(* PLC project mtcs_m1, Institute of Astronomy Onto 0.0.1 *)
(* stored: creationDateTime 2024-10-22T16:57:18.797943, modificationDateTime 2024-10-22T16:57:18.797943 *)

TYPE M1Parts : STRUCT
  inclinometer : M1Inclinometer;  (* Inclinometer *)
  radialSupport : M1RadialSupport;  (* Radial support *)
  axialSupport : M1AxialSupport;  (* Axial support *)
  io : M1M2IO;  (* I/O modules *)
  configManager : ConfigManager;  (* The config manager (to load/save/activate configuration data) *)
END_STRUCT;
END_TYPE

TYPE M1RadialSupportParts : STRUCT
  vacuumRelay : SimpleRelay;  (* Switch Radial vacuum ON to retract the radial pads during mirror manipulations. *)
END_STRUCT;
END_TYPE

TYPE M1M2IOParts : STRUCT
  COU : EtherCatDevice;
  AI1 : EtherCatDevice;
  AI2 : EtherCatDevice;
  AI3 : EtherCatDevice;
  AO1 : EtherCatDevice;
  DO1 : EtherCatDevice;
  RES1 : EtherCatDevice;
  RES2 : EtherCatDevice;
  RES3 : EtherCatDevice;
  PWR1 : EtherCatDevice;
  SSI1 : EtherCatDevice;
  AI4 : EtherCatDevice;
  INC1 : EtherCatDevice;
  P5V1 : EtherCatDevice;
  DO2 : EtherCatDevice;
  DO3 : EtherCatDevice;
  RE1 : EtherCatDevice;
END_STRUCT;
END_TYPE

TYPE M1Processes : STRUCT
  initialize : Process;  (* Start initializing *)
  lock : Process;  (* Lock the system *)
  unlock : Process;  (* Unlock the system *)
  changeOperatingState : ChangeOperatingStateProcess;  (* Change the operating state (e.g. AUTO, MANUAL, ...) *)
END_STRUCT;
END_TYPE

TYPE M1RadialSupportProcesses : STRUCT
  changePressureSetpoint : ChangeSetpointProcess;  (* Change a pressure setpoint, in Bar *)
  changePressureSetpointState : ChangeOperatingStateProcess;  (* Change the operating state of the pressure setpoint only *)
END_STRUCT;
END_TYPE

TYPE M1AxialSupportProcesses : STRUCT
  changePressureSetpoint : ChangeSetpointProcess;  (* Change a pressure setpoint, in Bar *)
  changePressureSetpointState : ChangeOperatingStateProcess;  (* Change the operating state of the pressure setpoint only *)
END_STRUCT;
END_TYPE

TYPE M1Statuses : STRUCT
  initializationStatus : InitializationStatus;
  healthStatus : HealthStatus;
  busyStatus : BusyStatus;
  operatingStatus : OperatingStatus;
END_STRUCT;
END_TYPE

TYPE M1InclinometerStatuses : STRUCT
  healthStatus : HealthStatus;  (* Is the inclinometer elevation trustworthy? *)
END_STRUCT;
END_TYPE

TYPE M1RadialSupportStatuses : STRUCT
  pressureSetpointStatus : OperatingStatus;  (* Operating status of the radial pressure setpoint *)
  healthStatus : HealthStatus;
  busyStatus : BusyStatus;
END_STRUCT;
END_TYPE

TYPE M1AxialSupportStatuses : STRUCT
  pressureSetpointStatus : OperatingStatus;  (* Operating status of the radial pressure setpoint *)
  healthStatus : HealthStatus;
  busyStatus : BusyStatus;
END_STRUCT;
END_TYPE

TYPE M1M2IOStatuses : STRUCT
  healthStatus : HealthStatus;  (* Is the I/O in a healthy state? *)
END_STRUCT;
END_TYPE

TYPE M1Config : STRUCT
  radialSupport : M1RadialSupportConfig;  (* Radial support *)
  axialSupport : M1AxialSupportConfig;  (* Axial support *)
  pneumaticSupplySensorFullScale : LREAL;  (* Sensor full scale range, in Bar *)
  pneumaticSupplyPressure : MeasurementConfig;  (* Pneumatic supply pressure config, in Bar *)
  inclinometerVoltage : MeasurementConfig;  (* Inclinometer voltage measuremennt config, in Volts *)
END_STRUCT;
END_TYPE

TYPE M1RadialSupportConfig : STRUCT
  regulatorPressure : MeasurementConfig;  (* Regulator pressure config, in Bar *)
  mirrorPressure : MeasurementConfig;  (* Regulator pressure config, in Bar *)
  regulatorPressureSensorFullScale : LREAL;  (* Sensor full scale range, in Bar *)
  mirrorPressureSensorFullScale : LREAL;  (* Sensor full scale range, in Bar *)
  correctionCoefficient : LREAL;  (* Correction coefficient for radial pressure *)
  controllerLimitMax : LREAL;  (* Maximum output of the controller, in Bar *)
  controllerLimitMin : LREAL;  (* Minimum output of the controller, in Bar *)
  pressureRegulatorRange : LREAL;  (* Pressure regulator range, in Bar *)
END_STRUCT;
END_TYPE

TYPE M1AxialSupportConfig : STRUCT
  regulatorPressure : MeasurementConfig;  (* Regulator pressure config, in Bar *)
  mirrorPressure : MeasurementConfig;  (* Regulator pressure config, in Bar *)
  mirrorSouthForce : MeasurementConfig;  (* Mirror south force config, in decaNewton *)
  mirrorNorthEastForce : MeasurementConfig;  (* Mirror north east force config, in decaNewton *)
  mirrorNorthWestForce : MeasurementConfig;  (* Mirror north west force config, in decaNewton *)
  mirrorAverageForce : MeasurementConfig;  (* Mirror moving average force config, in decaNewton *)
  regulatorPressureSensorFullScale : LREAL;  (* Sensor full scale range, in Bar *)
  mirrorPressureSensorFullScale : LREAL;  (* Sensor full scale range, in Bar *)
  correctionCoefficient : LREAL;  (* Correction coefficient for axial pressure *)
  controllerKp : LREAL;  (* Proportional factor (gain) of the PI controller *)
  controllerTn : LREAL;  (* Integral time factor of the PI controller. in seconds *)
  controllerLimitMax : LREAL;  (* Maximum output of the controller, in Bar *)
  controllerLimitMin : LREAL;  (* Minimum output of the controller, in Bar *)
  pressureRegulatorRange : LREAL;  (* Pressure regulator range, in Bar *)
END_STRUCT;
END_TYPE

FUNCTION_BLOCK SM_M1
  VAR_INPUT
    {attribute 'OPC.UA.DA' := '1'}
    {attribute 'OPC.UA.DA.Access' := '1'}
    editableConfig : M1Config;  (* Editable configuration of the M1 subsystem *)
  END_VAR
  VAR_OUTPUT
    {attribute 'OPC.UA.DA' := '1'}
    {attribute 'OPC.UA.DA.Access' := '1'}
    actualStatus : STRING;  (* Current status description *)
    previousStatus : STRING;  (* Previous status description *)
    {attribute 'OPC.UA.DA' := '1'}
    {attribute 'OPC.UA.DA.Access' := '1'}
    config : M1Config;  (* Active configuration of the M1 subsystem *)
    {attribute 'OPC.UA.DA' := '1'}
    {attribute 'OPC.UA.DA.Access' := '1'}
    pneumaticSupplyPressure : PressureMeasurement;  (* Pressure measurement of the pneumatic supply *)
    statuses : M1Statuses;  (* Statuses of the state machine *)
    parts : M1Parts;  (* Parts of the state machine *)
    processes : M1Processes;  (* Processes of the state machine *)
  END_VAR
  VAR_IN_OUT
    {attribute 'OPC.UA.DA' := '0'}
    operatorStatus : OperatorStatus;  (* Shared operator status *)
    {attribute 'OPC.UA.DA' := '0'}
    tubeAngleMeasurement : TelemetryAccelerometer;  (* Accelerometer box angle measurement *)
  END_VAR

            pneumaticSupplyPressure(
    config := config.pneumaticSupplyPressure,
    conversionFactor := config.pneumaticSupplySensorFullScale / 32768.0);
parts.inclinometer( config := config.inclinometerVoltage );
parts.radialSupport(
    config := config.radialSupport,
    inclinometer := parts.inclinometer,
    operatorStatus := operatorStatus,
    operatingStatus := statuses.operatingStatus);
parts.axialSupport(
    config := config.axialSupport,
    inclinometer := parts.inclinometer,
    operatorStatus := operatorStatus,
    operatingStatus := statuses.operatingStatus,
    tubeAngle := tubeAngleMeasurement.averageYAngle);
parts.io();
parts.configManager( isEnabled := operatorStatus.tech );
statuses.initializationStatus();
statuses.healthStatus(
    isGood := parts.radialSupport.statuses.healthStatus.isGood AND (parts.axialSupport.statuses.healthStatus.isGood AND (parts.io.statuses.healthStatus.isGood AND parts.configManager.statuses.healthStatus.isGood)),
    hasWarning := parts.radialSupport.statuses.healthStatus.hasWarning OR (parts.axialSupport.statuses.healthStatus.hasWarning OR (parts.io.statuses.healthStatus.hasWarning OR parts.configManager.statuses.healthStatus.hasWarning)));
statuses.busyStatus( isBusy := statuses.initializationStatus.initializing OR (parts.radialSupport.statuses.busyStatus.busy OR (parts.axialSupport.statuses.busyStatus.busy OR parts.configManager.statuses.busyStatus.busy)) );
statuses.operatingStatus( superState := statuses.initializationStatus.initialized );
processes.initialize( isEnabled := statuses.initializationStatus.shutdown OR (statuses.initializationStatus.initializingFailed OR statuses.initializationStatus.initialized) );
processes.lock( isEnabled := operatorStatus.tech AND statuses.initializationStatus.initialized );
processes.unlock( isEnabled := operatorStatus.tech AND statuses.initializationStatus.locked );
processes.changeOperatingState( isEnabled := statuses.busyStatus.idle AND (statuses.initializationStatus.initialized AND operatorStatus.tech) );

          

{attribute 'TcRpcEnable' := '1'}
METHOD initialize : RequestResults
                  initialize := THIS^.processes.initialize.request();

                
END_METHOD

{attribute 'TcRpcEnable' := '1'}
METHOD lock : RequestResults
                  lock := THIS^.processes.lock.request();

                
END_METHOD

{attribute 'TcRpcEnable' := '1'}
METHOD unlock : RequestResults
                  unlock := THIS^.processes.unlock.request();

                
END_METHOD

{attribute 'TcRpcEnable' := '1'}
METHOD changeOperatingState : RequestResults
  VAR_INPUT
    state : OperatingStates;
  END_VAR
                  changeOperatingState := THIS^.processes.changeOperatingState.request( state := state );

                
END_METHOD

{attribute 'TcRpcEnable' := '1'}
METHOD _log : BOOL
  VAR_INPUT
    name : STRING;  (* Name of this function block instance *)
  END_VAR
  VAR_IN_OUT
    buffer : LogBuffer;  (* Buffer to write all logging to *)
  END_VAR
  VAR
    subBuffer : LogBuffer;  (* Temporary buffer to write logging by parts (sub-statemachines) to *)
  END_VAR
                  THIS^.parts.inclinometer._log(
    name := 'inclinometer',
    buffer := subBuffer);
THIS^.parts.radialSupport._log(
    name := 'radialSupport',
    buffer := subBuffer);
THIS^.parts.axialSupport._log(
    name := 'axialSupport',
    buffer := subBuffer);
THIS^.parts.io._log(
    name := 'io',
    buffer := subBuffer);
THIS^.parts.configManager._log(
    name := 'configManager',
    buffer := subBuffer);
THIS^.processes.initialize._log(
    name := 'processes.initialize',
    buffer := subBuffer);
THIS^.processes.lock._log(
    name := 'processes.lock',
    buffer := subBuffer);
THIS^.processes.unlock._log(
    name := 'processes.unlock',
    buffer := subBuffer);
THIS^.processes.changeOperatingState._log(
    name := 'processes.changeOperatingState',
    buffer := subBuffer);
LOGGER(
    name := name,
    actualStatus := THIS^.actualStatus,
    previousStatus := THIS^.previousStatus,
    buffer := buffer,
    subBuffer := subBuffer,
    pHealthStatus := ADR(THIS^.statuses.healthStatus),
    pBusyStatus := ADR(THIS^.statuses.busyStatus));

                
END_METHOD
END_FUNCTION_BLOCK

FUNCTION_BLOCK SM_M1Inclinometer
  VAR_INPUT
    {attribute 'OPC.UA.DA' := '1'}
    {attribute 'OPC.UA.DA.Access' := '1'}
    voltageMeasurement : VoltageMeasurement;  (* Measured voltage *)
  END_VAR
  VAR_OUTPUT
    {attribute 'OPC.UA.DA' := '1'}
    {attribute 'OPC.UA.DA.Access' := '1'}
    actualStatus : STRING;  (* Current status description *)
    previousStatus : STRING;  (* Previous status description *)
    {attribute 'OPC.UA.DA' := '1'}
    {attribute 'OPC.UA.DA.Access' := '1'}
    actualElevation : AngularPosition;  (* Elevation actual value *)
    {attribute 'OPC.UA.DA' := '1'}
    {attribute 'OPC.UA.DA.Access' := '1'}
    averageElevation : AngularPosition;  (* Elevation average value *)
    statuses : M1InclinometerStatuses;  (* Statuses of the state machine *)
  END_VAR
  VAR_IN_OUT
    {attribute 'OPC.UA.DA' := '0'}
    config : MeasurementConfig;  (* Reference to the config *)
  END_VAR

            voltageMeasurement(
    config := config,
    conversionFactor := 10.0 / 32768.0);
statuses.healthStatus(
    isGood := voltageMeasurement.statuses.healthStatus.isGood,
    hasWarning := voltageMeasurement.statuses.healthStatus.hasWarning);

          

{attribute 'TcRpcEnable' := '1'}
METHOD _log : BOOL
  VAR_INPUT
    name : STRING;  (* Name of this function block instance *)
  END_VAR
  VAR_IN_OUT
    buffer : LogBuffer;  (* Buffer to write all logging to *)
  END_VAR
  VAR
    subBuffer : LogBuffer;  (* Temporary buffer to write logging by parts (sub-statemachines) to *)
  END_VAR
                  LOGGER(
    name := name,
    actualStatus := THIS^.actualStatus,
    previousStatus := THIS^.previousStatus,
    buffer := buffer,
    subBuffer := subBuffer,
    pHealthStatus := ADR(THIS^.statuses.healthStatus));

                
END_METHOD
END_FUNCTION_BLOCK

FUNCTION_BLOCK SM_M1RadialSupport
  VAR_INPUT
    {attribute 'OPC.UA.DA' := '0'}
    pressureSetpointOutput AT %Q* : INT;  (* Output value *)
  END_VAR
  VAR_OUTPUT
    {attribute 'OPC.UA.DA' := '1'}
    {attribute 'OPC.UA.DA.Access' := '1'}
    actualStatus : STRING;  (* Current status description *)
    previousStatus : STRING;  (* Previous status description *)
    {attribute 'OPC.UA.DA' := '1'}
    {attribute 'OPC.UA.DA.Access' := '1'}
    regulatorPressure : PressureMeasurement;  (* Pressure measurement at the regulator *)
    {attribute 'OPC.UA.DA' := '1'}
    {attribute 'OPC.UA.DA.Access' := '1'}
    mirrorPressure : PressureMeasurement;  (* Pressure measurement at the mirror *)
    {attribute 'OPC.UA.DA' := '1'}
    {attribute 'OPC.UA.DA.Access' := '1'}
    actualPressureSetpoint : Pressure;  (* Pressure setpoint actually used *)
    {attribute 'OPC.UA.DA' := '1'}
    {attribute 'OPC.UA.DA.Access' := '1'}
    autoPressureSetpoint : Pressure;  (* Pressure setpoint in AUTO mode *)
    {attribute 'OPC.UA.DA' := '1'}
    {attribute 'OPC.UA.DA.Access' := '1'}
    manualPressureSetpoint : Pressure;  (* Pressure setpoint in MANUAL mode *)
    statuses : M1RadialSupportStatuses;  (* Statuses of the state machine *)
    parts : M1RadialSupportParts;  (* Parts of the state machine *)
    processes : M1RadialSupportProcesses;  (* Processes of the state machine *)
  END_VAR
  VAR_IN_OUT
    {attribute 'OPC.UA.DA' := '0'}
    config : M1RadialSupportConfig;
    {attribute 'OPC.UA.DA' := '0'}
    inclinometer : M1Inclinometer;
    {attribute 'OPC.UA.DA' := '0'}
    operatorStatus : OperatorStatus;
    {attribute 'OPC.UA.DA' := '0'}
    operatingStatus : OperatingStatus;
  END_VAR

            regulatorPressure(
    config := config.regulatorPressure,
    conversionFactor := config.regulatorPressureSensorFullScale / 32768.0);
mirrorPressure(
    config := config.mirrorPressure,
    conversionFactor := config.mirrorPressureSensorFullScale / 32768.0);
parts.vacuumRelay( isEnabled := statuses.busyStatus.idle AND (operatingStatus.manual AND operatorStatus.tech) );
statuses.pressureSetpointStatus();
statuses.healthStatus(
    isGood := (processes.changePressureSetpointState.statuses.healthStatus.isGood AND (processes.changePressureSetpoint.statuses.healthStatus.isGood AND regulatorPressure.statuses.healthStatus.isGood)) AND (mirrorPressure.statuses.healthStatus.isGood OR mirrorPressure.statuses.enabledStatus.disabled),
    hasWarning := (processes.changePressureSetpointState.statuses.healthStatus.hasWarning OR (processes.changePressureSetpoint.statuses.healthStatus.hasWarning OR (regulatorPressure.statuses.healthStatus.hasWarning OR mirrorPressure.statuses.healthStatus.hasWarning))) OR parts.vacuumRelay.digitalOutput);
statuses.busyStatus( isBusy := processes.changePressureSetpointState.statuses.busyStatus.busy OR (processes.changePressureSetpoint.statuses.busyStatus.busy OR parts.vacuumRelay.statuses.busyStatus.busy) );
processes.changePressureSetpoint( isEnabled := parts.vacuumRelay.isEnabled );
processes.changePressureSetpointState( isEnabled := parts.vacuumRelay.isEnabled );

          

{attribute 'TcRpcEnable' := '1'}
METHOD changePressureSetpoint : RequestResults
  VAR_INPUT
    setpoint : LREAL;
  END_VAR
                  changePressureSetpoint := THIS^.processes.changePressureSetpoint.request( setpoint := setpoint );

                
END_METHOD

{attribute 'TcRpcEnable' := '1'}
METHOD changePressureSetpointState : RequestResults
  VAR_INPUT
    state : OperatingStates;
  END_VAR
                  changePressureSetpointState := THIS^.processes.changePressureSetpointState.request( state := state );

                
END_METHOD

{attribute 'TcRpcEnable' := '1'}
METHOD _log : BOOL
  VAR_INPUT
    name : STRING;  (* Name of this function block instance *)
  END_VAR
  VAR_IN_OUT
    buffer : LogBuffer;  (* Buffer to write all logging to *)
  END_VAR
  VAR
    subBuffer : LogBuffer;  (* Temporary buffer to write logging by parts (sub-statemachines) to *)
  END_VAR
                  THIS^.parts.vacuumRelay._log(
    name := 'vacuumRelay',
    buffer := subBuffer);
THIS^.processes.changePressureSetpoint._log(
    name := 'processes.changePressureSetpoint',
    buffer := subBuffer);
THIS^.processes.changePressureSetpointState._log(
    name := 'processes.changePressureSetpointState',
    buffer := subBuffer);
LOGGER(
    name := name,
    actualStatus := THIS^.actualStatus,
    previousStatus := THIS^.previousStatus,
    buffer := buffer,
    subBuffer := subBuffer,
    pHealthStatus := ADR(THIS^.statuses.healthStatus),
    pBusyStatus := ADR(THIS^.statuses.busyStatus));

                
END_METHOD
END_FUNCTION_BLOCK

FUNCTION_BLOCK SM_M1AxialSupport
  VAR_INPUT
    {attribute 'OPC.UA.DA' := '0'}
    pressureSetpointOutput AT %Q* : INT;  (* Output value *)
  END_VAR
  VAR_OUTPUT
    {attribute 'OPC.UA.DA' := '1'}
    {attribute 'OPC.UA.DA.Access' := '1'}
    actualStatus : STRING;  (* Current status description *)
    previousStatus : STRING;  (* Previous status description *)
    {attribute 'OPC.UA.DA' := '1'}
    {attribute 'OPC.UA.DA.Access' := '1'}
    regulatorPressure : PressureMeasurement;  (* Pressure measurement at the regulator *)
    {attribute 'OPC.UA.DA' := '1'}
    {attribute 'OPC.UA.DA.Access' := '1'}
    mirrorPressure : PressureMeasurement;  (* Pressure measurement at the mirror *)
    {attribute 'OPC.UA.DA' := '1'}
    {attribute 'OPC.UA.DA.Access' := '1'}
    mirrorSouthForce : ForceMeasurement;  (* Force measurement South (SO) *)
    {attribute 'OPC.UA.DA' := '1'}
    {attribute 'OPC.UA.DA.Access' := '1'}
    mirrorNorthEastForce : ForceMeasurement;  (* Force measurement North East (NE) *)
    {attribute 'OPC.UA.DA' := '1'}
    {attribute 'OPC.UA.DA.Access' := '1'}
    mirrorNorthWestForce : ForceMeasurement;  (* Force measurement North West (NW) *)
    {attribute 'OPC.UA.DA' := '1'}
    {attribute 'OPC.UA.DA.Access' := '1'}
    mirrorAverageForce : ForceMeasurement;  (* Average of SO, NE and NW *)
    {attribute 'OPC.UA.DA' := '1'}
    {attribute 'OPC.UA.DA.Access' := '1'}
    actualPressureSetpoint : Pressure;  (* Pressure setpoint actually used *)
    {attribute 'OPC.UA.DA' := '1'}
    {attribute 'OPC.UA.DA.Access' := '1'}
    autoPressureSetpoint : Pressure;  (* Pressure setpoint in AUTO mode *)
    {attribute 'OPC.UA.DA' := '1'}
    {attribute 'OPC.UA.DA.Access' := '1'}
    manualPressureSetpoint : Pressure;  (* Pressure setpoint in MANUAL mode *)
    {attribute 'OPC.UA.DA' := '1'}
    {attribute 'OPC.UA.DA.Access' := '1'}
    controllerSetpoint : Force;  (* Force setpoint of the controller *)
    statuses : M1AxialSupportStatuses;  (* Statuses of the state machine *)
    processes : M1AxialSupportProcesses;  (* Processes of the state machine *)
  END_VAR
  VAR_IN_OUT
    {attribute 'OPC.UA.DA' := '0'}
    config : M1AxialSupportConfig;
    {attribute 'OPC.UA.DA' := '0'}
    inclinometer : M1Inclinometer;
    {attribute 'OPC.UA.DA' := '0'}
    operatorStatus : OperatorStatus;
    {attribute 'OPC.UA.DA' := '0'}
    operatingStatus : OperatingStatus;
    {attribute 'OPC.UA.DA' := '0'}
    tubeAngle : AngularPosition;
  END_VAR

            regulatorPressure(
    config := config.regulatorPressure,
    conversionFactor := config.regulatorPressureSensorFullScale / 32768.0);
mirrorPressure(
    config := config.mirrorPressure,
    conversionFactor := config.mirrorPressureSensorFullScale / 32768.0);
mirrorSouthForce(
    config := config.mirrorSouthForce,
    conversionFactor := (-200.0 * 20.0) / 2147483648.0);
mirrorNorthEastForce(
    config := config.mirrorNorthEastForce,
    conversionFactor := (-200.0 * 20.0) / 2147483648.0);
mirrorNorthWestForce(
    config := config.mirrorNorthWestForce,
    conversionFactor := (-200.0 * 20.0) / 2147483648.0);
mirrorAverageForce(
    config := config.mirrorAverageForce,
    conversionFactor := (-200.0 * 20.0) / 2147483648.0);
statuses.pressureSetpointStatus();
statuses.healthStatus(
    isGood := (processes.changePressureSetpointState.statuses.healthStatus.isGood AND (processes.changePressureSetpoint.statuses.healthStatus.isGood AND (regulatorPressure.statuses.healthStatus.isGood AND mirrorAverageForce.statuses.healthStatus.isGood))) AND (mirrorPressure.statuses.healthStatus.isGood OR mirrorPressure.statuses.enabledStatus.disabled),
    hasWarning := processes.changePressureSetpointState.statuses.healthStatus.hasWarning OR (processes.changePressureSetpoint.statuses.healthStatus.hasWarning OR (regulatorPressure.statuses.healthStatus.hasWarning OR (mirrorPressure.statuses.healthStatus.hasWarning OR mirrorAverageForce.statuses.healthStatus.hasWarning))));
statuses.busyStatus( isBusy := processes.changePressureSetpointState.statuses.busyStatus.busy OR processes.changePressureSetpoint.statuses.busyStatus.busy );
processes.changePressureSetpoint( isEnabled := statuses.busyStatus.idle AND (operatingStatus.manual AND operatorStatus.tech) );
processes.changePressureSetpointState( isEnabled := statuses.busyStatus.idle AND (operatingStatus.manual AND operatorStatus.tech) );

          

{attribute 'TcRpcEnable' := '1'}
METHOD changePressureSetpoint : RequestResults
  VAR_INPUT
    setpoint : LREAL;
  END_VAR
                  changePressureSetpoint := THIS^.processes.changePressureSetpoint.request( setpoint := setpoint );

                
END_METHOD

{attribute 'TcRpcEnable' := '1'}
METHOD changePressureSetpointState : RequestResults
  VAR_INPUT
    state : OperatingStates;
  END_VAR
                  changePressureSetpointState := THIS^.processes.changePressureSetpointState.request( state := state );

                
END_METHOD

{attribute 'TcRpcEnable' := '1'}
METHOD _log : BOOL
  VAR_INPUT
    name : STRING;  (* Name of this function block instance *)
  END_VAR
  VAR_IN_OUT
    buffer : LogBuffer;  (* Buffer to write all logging to *)
  END_VAR
  VAR
    subBuffer : LogBuffer;  (* Temporary buffer to write logging by parts (sub-statemachines) to *)
  END_VAR
                  THIS^.processes.changePressureSetpoint._log(
    name := 'processes.changePressureSetpoint',
    buffer := subBuffer);
THIS^.processes.changePressureSetpointState._log(
    name := 'processes.changePressureSetpointState',
    buffer := subBuffer);
LOGGER(
    name := name,
    actualStatus := THIS^.actualStatus,
    previousStatus := THIS^.previousStatus,
    buffer := buffer,
    subBuffer := subBuffer,
    pHealthStatus := ADR(THIS^.statuses.healthStatus),
    pBusyStatus := ADR(THIS^.statuses.busyStatus));

                
END_METHOD
END_FUNCTION_BLOCK

FUNCTION_BLOCK SM_M1M2IO
  VAR_OUTPUT
    {attribute 'OPC.UA.DA' := '1'}
    {attribute 'OPC.UA.DA.Access' := '1'}
    actualStatus : STRING;  (* Current status description *)
    previousStatus : STRING;  (* Previous status description *)
    statuses : M1M2IOStatuses;  (* Statuses of the state machine *)
    parts : M1M2IOParts;  (* Parts of the state machine *)
  END_VAR

            parts.COU(
    id := 'M1M2:COU',
    typeId := 'EK1101');
parts.AI1(
    id := 'M1M2:AI1',
    typeId := 'EL3102');
parts.AI2(
    id := 'M1M2:AI2',
    typeId := 'EL3204');
parts.AI3(
    id := 'M1M2:AI3',
    typeId := 'EL3204');
parts.AO1(
    id := 'M1M2:AO1',
    typeId := 'EL4022');
parts.DO1(
    id := 'M1M2:DO1',
    typeId := 'EL2024');
parts.RES1(
    id := 'M1M2:RES1',
    typeId := 'EL3351');
parts.RES2(
    id := 'M1M2:RES2',
    typeId := 'EL3351');
parts.RES3(
    id := 'M1M2:RES3',
    typeId := 'EL3351');
parts.PWR1(
    id := 'M1M2:PWR1',
    typeId := 'EL9410');
parts.SSI1(
    id := 'M1M2:SSI1',
    typeId := 'EL5001');
parts.AI4(
    id := 'M1M2:AI4',
    typeId := 'EL3164');
parts.INC1(
    id := 'M1M2:INC1',
    typeId := 'ES5101');
parts.P5V1(
    id := 'M1M2:P5V1',
    typeId := 'EL9505');
parts.DO2(
    id := 'M1M2:DO2',
    typeId := 'EL2124');
parts.DO3(
    id := 'M1M2:DO3',
    typeId := 'EL2124');
parts.RE1(
    id := 'M1M2:RE1',
    typeId := 'EL2622');
statuses.healthStatus( isGood := parts.COU.statuses.healthStatus.isGood AND (parts.AI1.statuses.healthStatus.isGood AND (parts.AI2.statuses.healthStatus.isGood AND (parts.AI3.statuses.healthStatus.isGood AND (parts.AO1.statuses.healthStatus.isGood AND (parts.DO1.statuses.healthStatus.isGood AND (parts.RES1.statuses.healthStatus.isGood AND (parts.RES2.statuses.healthStatus.isGood AND (parts.RES3.statuses.healthStatus.isGood AND (parts.PWR1.statuses.healthStatus.isGood AND (parts.SSI1.statuses.healthStatus.isGood AND (parts.AI4.statuses.healthStatus.isGood AND (parts.INC1.statuses.healthStatus.isGood AND (parts.P5V1.statuses.healthStatus.isGood AND (parts.DO2.statuses.healthStatus.isGood AND (parts.DO3.statuses.healthStatus.isGood AND parts.RE1.statuses.healthStatus.isGood))))))))))))))) );

          

{attribute 'TcRpcEnable' := '1'}
METHOD _log : BOOL
  VAR_INPUT
    name : STRING;  (* Name of this function block instance *)
  END_VAR
  VAR_IN_OUT
    buffer : LogBuffer;  (* Buffer to write all logging to *)
  END_VAR
  VAR
    subBuffer : LogBuffer;  (* Temporary buffer to write logging by parts (sub-statemachines) to *)
  END_VAR
                  THIS^.parts.COU._log(
    name := 'COU',
    buffer := subBuffer);
THIS^.parts.AI1._log(
    name := 'AI1',
    buffer := subBuffer);
THIS^.parts.AI2._log(
    name := 'AI2',
    buffer := subBuffer);
THIS^.parts.AI3._log(
    name := 'AI3',
    buffer := subBuffer);
THIS^.parts.AO1._log(
    name := 'AO1',
    buffer := subBuffer);
THIS^.parts.DO1._log(
    name := 'DO1',
    buffer := subBuffer);
THIS^.parts.RES1._log(
    name := 'RES1',
    buffer := subBuffer);
THIS^.parts.RES2._log(
    name := 'RES2',
    buffer := subBuffer);
THIS^.parts.RES3._log(
    name := 'RES3',
    buffer := subBuffer);
THIS^.parts.PWR1._log(
    name := 'PWR1',
    buffer := subBuffer);
THIS^.parts.SSI1._log(
    name := 'SSI1',
    buffer := subBuffer);
THIS^.parts.AI4._log(
    name := 'AI4',
    buffer := subBuffer);
THIS^.parts.INC1._log(
    name := 'INC1',
    buffer := subBuffer);
THIS^.parts.P5V1._log(
    name := 'P5V1',
    buffer := subBuffer);
THIS^.parts.DO2._log(
    name := 'DO2',
    buffer := subBuffer);
THIS^.parts.DO3._log(
    name := 'DO3',
    buffer := subBuffer);
THIS^.parts.RE1._log(
    name := 'RE1',
    buffer := subBuffer);
LOGGER(
    name := name,
    actualStatus := THIS^.actualStatus,
    previousStatus := THIS^.previousStatus,
    buffer := buffer,
    subBuffer := subBuffer,
    pHealthStatus := ADR(THIS^.statuses.healthStatus));

                
END_METHOD
END_FUNCTION_BLOCK
